TYPE T_Hash_Code : LWORD; END_TYPE

(* stored: Version 1.1.0.1, ProductVersion 3.1.4024.4
   DUT T_Hash_Code: Id {14092f63-7f0e-4841-a7df-63780e53fca2} *)
